(* Logix 5000 project; controller BOX_FORMING_LADDER_RS32_logixEmulate Emulate 5570 rev 32.11; software revision 32.00 *)

TASK MainTask (continuous, watchdog 500 ms) : MainProgram

MODULES
   Local : Emulate 5570 (ICP 2, rev 32.11)
      I_O : vendor 1 type 0 code 15 (ICP 3, rev 1.1, Output RPI 150 ms)
           Local:3:I   // Entradas Digitales del Controlador
           Local:3:O   // Salidas Digitales del Controlador
END_MODULES

TYPE Bloque_Instrucciones :   // Bloque de instrucciones
STRUCT
   MGSD : MOTION_INSTRUCTION;   // Arreglo donde serán almacenados los datos del bloque de función MGSD
   MGS : MOTION_INSTRUCTION;   // Arreglo donde serán almacenados los datos del bloque de función MGS
   MGSR : MOTION_INSTRUCTION;   // Arreglo donde serán almacenados los datos del bloque de función MGSR
   MAFR : MOTION_INSTRUCTION;   // Arreglo donde serán almacenados los datos del bloque de función MAFR
   MASR : MOTION_INSTRUCTION;   // Arreglo donde serán almacenados los datos del bloque de función MASR
   MSO : MOTION_INSTRUCTION;   // Arreglo donde serán almacenados los datos del bloque de función MSO
   MSF : MOTION_INSTRUCTION;   // Arreglo donde serán almacenados los datos del bloque de función MSF
   MAS : MOTION_INSTRUCTION[3];   // Arreglo donde serán almacenados los datos del bloque de función MAS
   MAH : MOTION_INSTRUCTION;   // Arreglo donde serán almacenados los datos del bloque de función MAH
   MAJ : MOTION_INSTRUCTION;   // Arreglo donde serán almacenados los datos del bloque de función MAJ
   MAG : MOTION_INSTRUCTION;   // Arreglo donde serán almacenados los datos del bloque de función MAG
   MAM : MOTION_INSTRUCTION[3];   // Arreglo donde serán almacenados los datos del bloque de función MAM
END_STRUCT
END_TYPE

VAR_GLOBAL   (* controller tags *)
   Conveyor_Belt : Bloque_Instrucciones := (MSO.FLAGS := -1577058304, MSO.EN := 1, MSO.DN := 1, MSO.STATE := 1, MSF.FLAGS := 33554432, MAS[0].FLAGS := 33554432, MAS[1].FLAGS := 33554432, MAS[2].FLAGS := 33554432, MAH.FLAGS := 33554432, MAJ.FLAGS := 570425344, MAJ.DN := 1, MAG.FLAGS := 570425344, MAG.DN := 1, MAM[0].FLAGS := 33554432, MAM[1].FLAGS := 33554432);
   Conveyor_Belt_Velocidad_Actual : REAL;   // Señal NX - Output
   DriveMSGD : MOTION_INSTRUCTION;   // Arreglo donde serán almacenados los datos del bloque de función MSGD
   Driver : Bloque_Instrucciones := (MGSD.FLAGS := 33554432, MGS.FLAGS := 33554432, MGSR.FLAGS := -1577058304, MGSR.EN := 1, MGSR.DN := 1, MAFR.FLAGS := 33554432, MASR.FLAGS := 33554432);
   DriverMAFR : MOTION_INSTRUCTION;   // Arreglo donde serán almacenados los datos del bloque de función MAFR
   DriverMASR : MOTION_INSTRUCTION;   // Arreglo donde serán almacenados los datos del bloque de función MASR
   DriverMGS : MOTION_INSTRUCTION;   // Arreglo donde serán almacenados los datos del bloque de función MGS
   DriverMGSD : MOTION_INSTRUCTION;   // Arreglo donde serán almacenados los datos del bloque de función MGSD
   DriverMGSR : MOTION_INSTRUCTION;   // Arreglo donde serán almacenados los datos del bloque de función MGSR
   DriverMSF : MOTION_INSTRUCTION;   // Arreglo donde serán almacenados los datos del bloque de función MSF
   DriverMSO : MOTION_INSTRUCTION;   // Arreglo donde serán almacenados los datos del bloque de función MSO
   Eje_X : Bloque_Instrucciones := (MSO.FLAGS := -1577058304, MSO.EN := 1, MSO.DN := 1, MSO.STATE := 1, MSF.FLAGS := 33554432, MAS[0].FLAGS := 33554432, MAS[1].FLAGS := 33554432, MAS[2].FLAGS := 33554432, MAH.FLAGS := 33554432, MAM[0].FLAGS := 33554432, MAM[1].FLAGS := 33554432, MAM[2].FLAGS := -1577058304, MAM[2].EN := 1, MAM[2].DN := 1);
   Eje_X_Posicion_Actual : REAL;   // Señal NX - Output
   Eje_Y : Bloque_Instrucciones := (MSO.FLAGS := -1577058304, MSO.EN := 1, MSO.DN := 1, MSO.STATE := 1, MSF.FLAGS := 33554432, MAS[0].FLAGS := 33554432, MAS[1].FLAGS := 33554432, MAS[2].FLAGS := 33554432, MAH.FLAGS := 33554432, MAM[0].FLAGS := 33554432, MAM[1].FLAGS := 33554432);
   Eje_Y_Posicion_Actual : REAL;   // Señal NX - Output
   Eje_Z : Bloque_Instrucciones := (MSO.FLAGS := -1577058304, MSO.EN := 1, MSO.DN := 1, MSO.STATE := 1, MSF.FLAGS := 33554432, MAS[0].FLAGS := 33554432, MAS[1].FLAGS := 33554432, MAS[2].FLAGS := 33554432, MAH.FLAGS := 33554432, MAJ.FLAGS := 637534208, MAJ.DN := 1, MAJ.IP := 1, MAG.FLAGS := 570425344, MAG.DN := 1, MAM[0].FLAGS := 33554432, MAM[1].FLAGS := 33554432);
   Eje_Z_Posicion_Actual : REAL;   // Señal NX - Output
   Fault_Reset : BOOL;
   Group_1 : MOTION_GROUP;
   Init : DINT;
   SENSOR_CAJA : BOOL;   // Señal NX - Ouput Indicator
   SPAWN_CAJA : BOOL;   // Señal NX - Output
   START_ALL : BOOL;   // BIT Destinado a la Habilitación del Sistema
   STOP_ALL : BOOL;   // BIT Destinado a la Parada del Sistema
   TESTIGO_START_ALL : ALIAS FOR Local:3:O.Data[0].0;
   TESTIGO_STOP_ALL : ALIAS FOR Local:3:O.Data[0].1;
   VIRTUAL_CONVEYOR_BELT : AXIS_VIRTUAL;   // Servomotor de la Banda Transportadora
   VIRTUAL_X_AXIS : AXIS_VIRTUAL;   // Servomotor del Eje X
   VIRTUAL_Y_AXIS : AXIS_VIRTUAL;   // Servomotor del Eje Y
   VIRTUAL_Z_AXIS : AXIS_VIRTUAL;   // Servomotor del Eje Z
END_VAR

PROGRAM MainProgram   (* main routine Main *)
VAR
   B0 : BOOL;   // Boxes Initialization Sync.
   C0 : BOOL;   // OK-INITIALIZATION
   C1 : BOOL;   // OK-CONVEYOR_BELT_IS_ON
   C2 : BOOL;   // OK-FORMADO_MOV_Y_Z
   C3 : BOOL;   // OK-FORMADO_MOV_X
   C4 : BOOL;   // OK-HOME_MOV_X_Y_Z
   C5 : BOOL;   // OK-RESET_PROCESS
   E0 : BOOL;   // INITIALIZATION
   E1 : BOOL;   // CONVEYOR_BELT_IS_ON
   E2 : BOOL;   // FORMADO_MOV_Y_Z
   E3 : BOOL;   // FORMADO_MOV_X
   E4 : BOOL;   // HOME_MOV_X_Y_Z
   E5 : BOOL;   // RESET_PROCESS
   F0 : BOOL;   // HOME_MOV_X: Transition Condition
   Fault_Reset : BOOL;   // Resetea todas las fallas/errores ocurridas en el Servo o el Driver
   H0 : BOOL;   // OK-HOME_MOV_Z: Home Flag [0]
   Servo_Off : BOOL;   // Botón físico que desabilita/desenergiza los servos
   Timer_Break_Forming : TIMER := (PRE := 400);   // Forming Break Time
   Timer_Break_Home : TIMER := (PRE := 400);   // Home Break Time
   Timer_Sensor : TIMER := (PRE := 8000);
END_VAR

ROUTINE A_Process_Setup   (* ladder *)
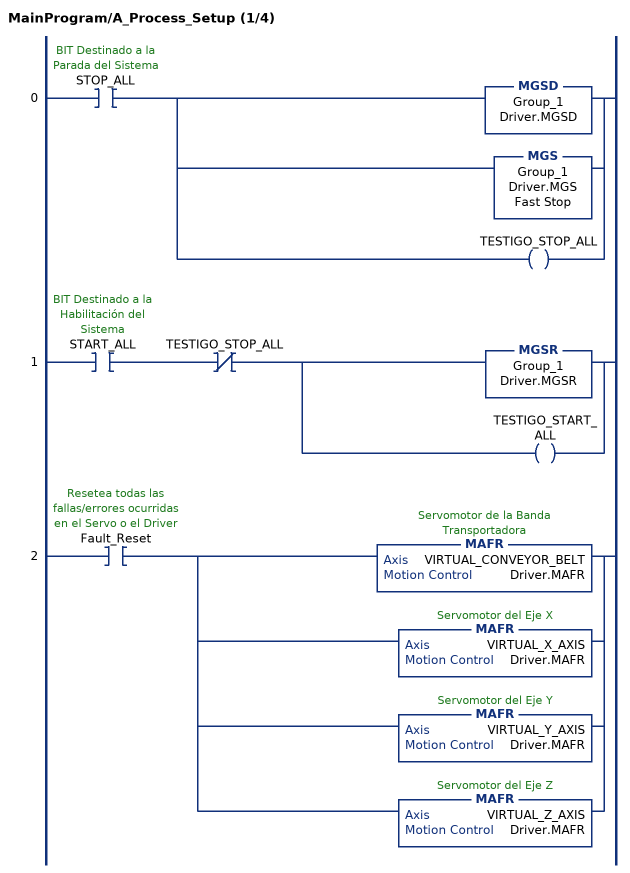
   0: XIC(STOP_ALL)[MGSD(Group_1,Driver.MGSD) ,MGS(Group_1,Driver.MGS,Fast Stop) ,OTE(TESTIGO_STOP_ALL) ];
   1: XIC(START_ALL)XIO(TESTIGO_STOP_ALL)[MGSR(Group_1,Driver.MGSR) ,OTE(TESTIGO_START_ALL) ];
   2: XIC(Fault_Reset)[MAFR(VIRTUAL_CONVEYOR_BELT,Driver.MAFR) ,MAFR(VIRTUAL_X_AXIS,Driver.MAFR) ,MAFR(VIRTUAL_Y_AXIS,Driver.MAFR) ,MAFR(VIRTUAL_Z_AXIS,Driver.MAFR) ];
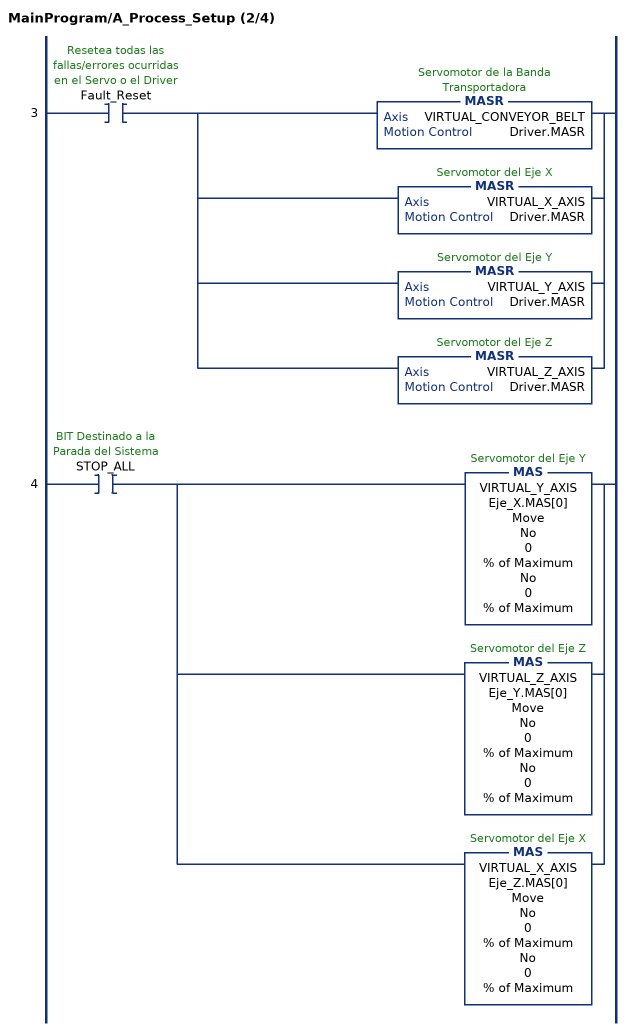
   3: XIC(Fault_Reset)[MASR(VIRTUAL_CONVEYOR_BELT,Driver.MASR) ,MASR(VIRTUAL_X_AXIS,Driver.MASR) ,MASR(VIRTUAL_Y_AXIS,Driver.MASR) ,MASR(VIRTUAL_Z_AXIS,Driver.MASR) ];
   4: XIC(STOP_ALL)[MAS(VIRTUAL_Y_AXIS,Eje_X.MAS[0],Move,No,0,% of Maximum,No,0,% of Maximum) ,MAS(VIRTUAL_Z_AXIS,Eje_Y.MAS[0],Move,No,0,% of Maximum,No,0,% of Maximum) ,MAS(VIRTUAL_X_AXIS,Eje_Z.MAS[0],Move,No,0,% of Maximum,No,0,% of Maximum) ];
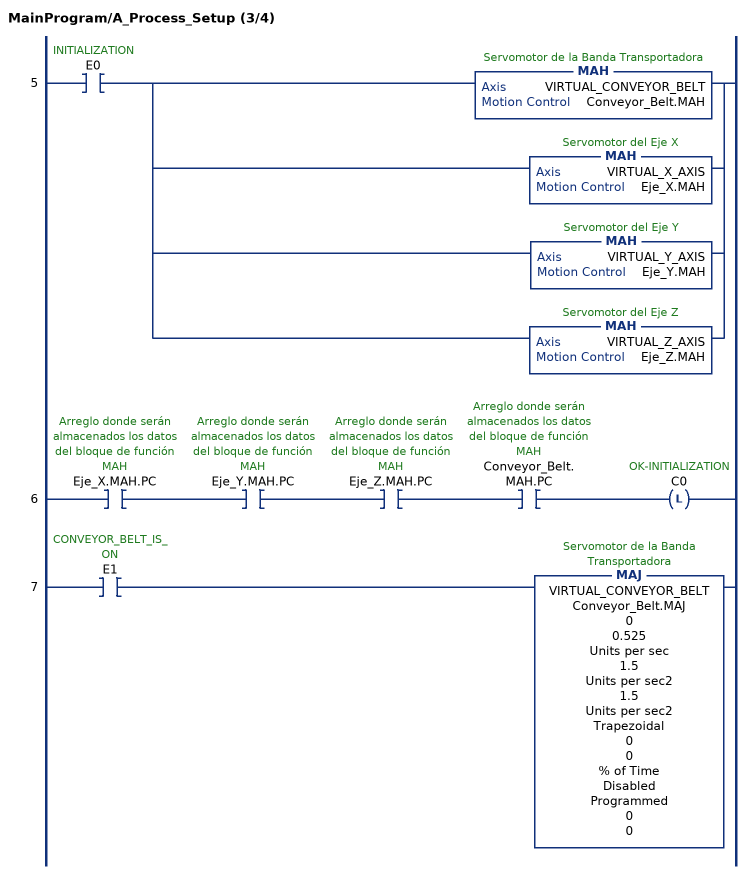
   5: XIC(E0)[MAH(VIRTUAL_CONVEYOR_BELT,Conveyor_Belt.MAH) ,MAH(VIRTUAL_X_AXIS,Eje_X.MAH) ,MAH(VIRTUAL_Y_AXIS,Eje_Y.MAH) ,MAH(VIRTUAL_Z_AXIS,Eje_Z.MAH) ];
   6: XIC(Eje_X.MAH.PC)XIC(Eje_Y.MAH.PC)XIC(Eje_Z.MAH.PC)XIC(Conveyor_Belt.MAH.PC)OTL(C0);
   7: XIC(E1)MAJ(VIRTUAL_CONVEYOR_BELT,Conveyor_Belt.MAJ,0,0.525,Units per sec,1.5,Units per sec2,1.5,Units per sec2,Trapezoidal,0,0,% of Time,Disabled,Programmed,0,0);
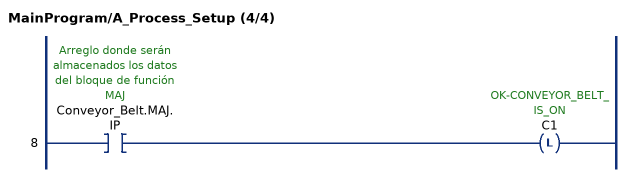
   8: XIC(Conveyor_Belt.MAJ.IP)OTL(C1);
END_ROUTINE

ROUTINE B_Process_Formado   (* ladder *)
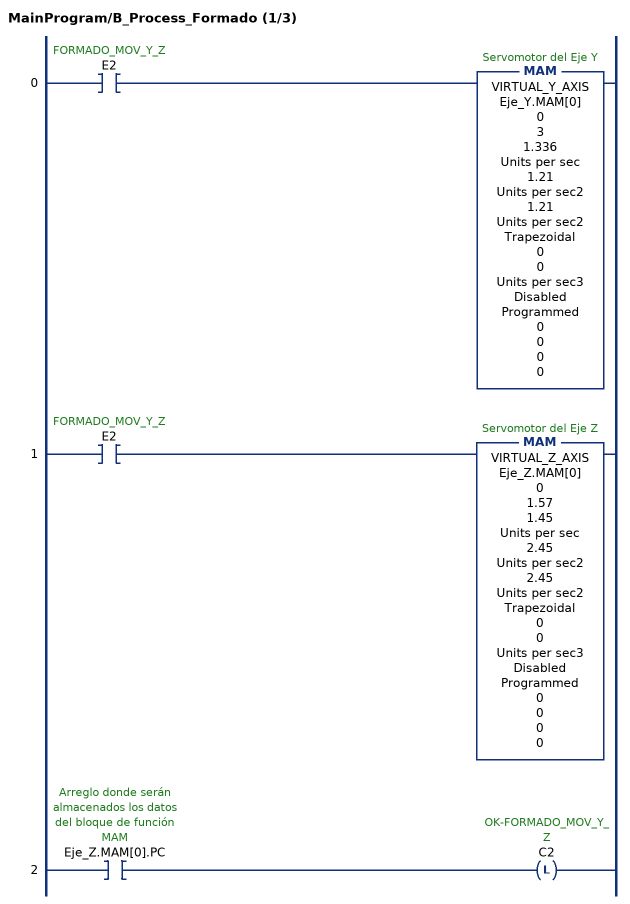
   0: XIC(E2)MAM(VIRTUAL_Y_AXIS,Eje_Y.MAM[0],0,3,1.336,Units per sec,1.21,Units per sec2,1.21,Units per sec2,Trapezoidal,0,0,Units per sec3,Disabled,Programmed,0,0,0,0);
   1: XIC(E2)MAM(VIRTUAL_Z_AXIS,Eje_Z.MAM[0],0,1.57,1.45,Units per sec,2.45,Units per sec2,2.45,Units per sec2,Trapezoidal,0,0,Units per sec3,Disabled,Programmed,0,0,0,0);
   2: XIC(Eje_Z.MAM[0].PC)OTL(C2);
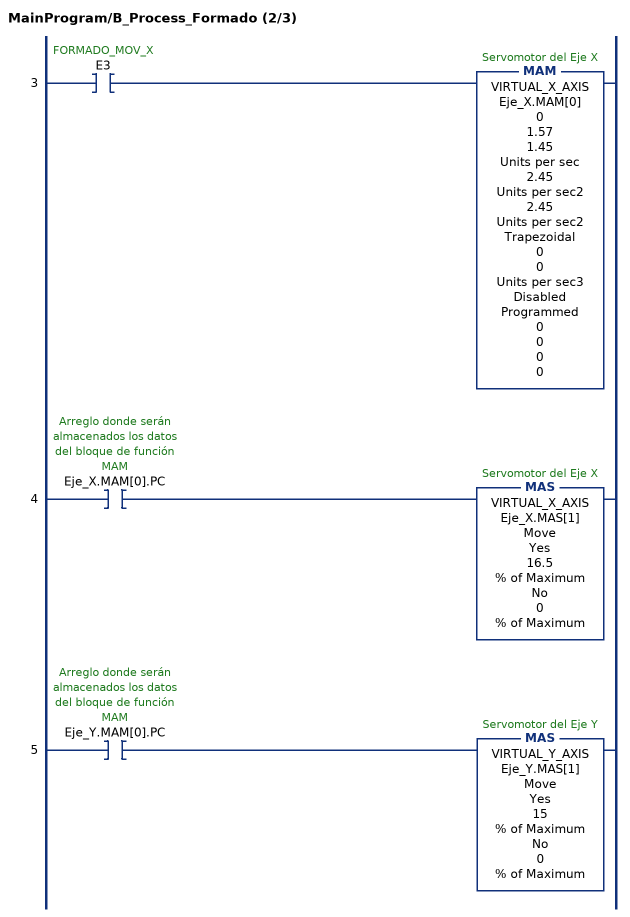
   3: XIC(E3)MAM(VIRTUAL_X_AXIS,Eje_X.MAM[0],0,1.57,1.45,Units per sec,2.45,Units per sec2,2.45,Units per sec2,Trapezoidal,0,0,Units per sec3,Disabled,Programmed,0,0,0,0);
   4: XIC(Eje_X.MAM[0].PC)MAS(VIRTUAL_X_AXIS,Eje_X.MAS[1],Move,Yes,16.5,% of Maximum,No,0,% of Maximum);
   5: XIC(Eje_Y.MAM[0].PC)MAS(VIRTUAL_Y_AXIS,Eje_Y.MAS[1],Move,Yes,15,% of Maximum,No,0,% of Maximum);
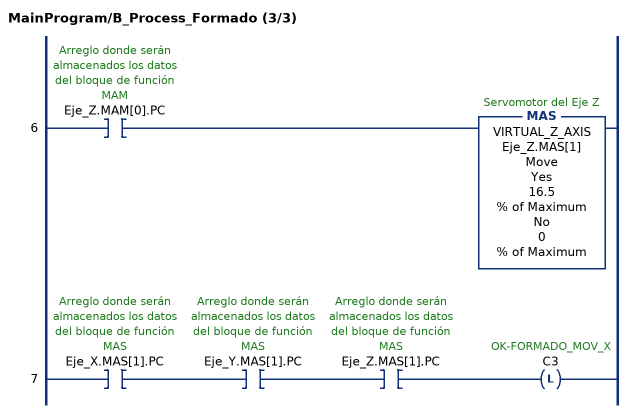
   6: XIC(Eje_Z.MAM[0].PC)MAS(VIRTUAL_Z_AXIS,Eje_Z.MAS[1],Move,Yes,16.5,% of Maximum,No,0,% of Maximum);
   7: XIC(Eje_X.MAS[1].PC)XIC(Eje_Y.MAS[1].PC)XIC(Eje_Z.MAS[1].PC)OTL(C3);
END_ROUTINE

ROUTINE C_Process_Home   (* ladder *)
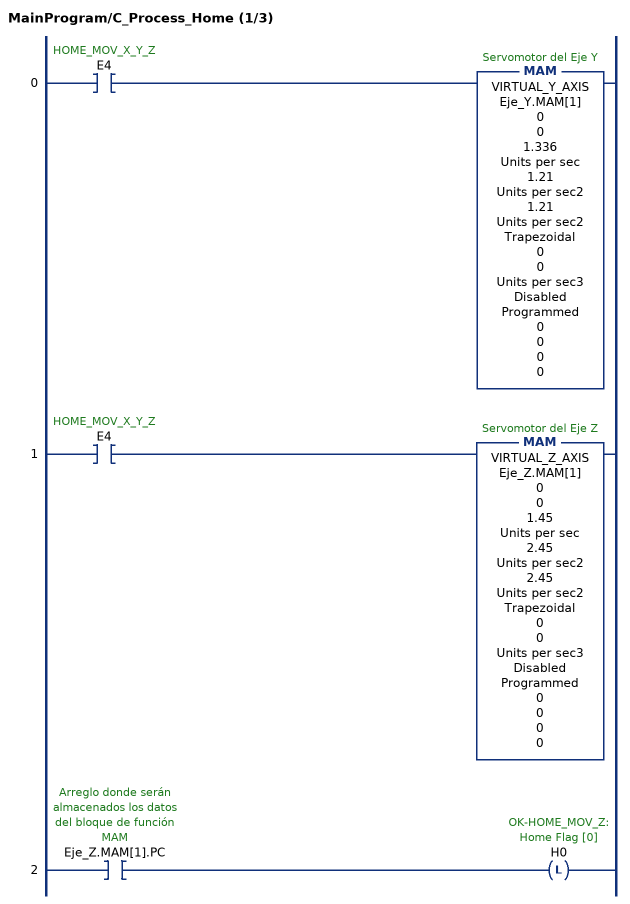
   0: XIC(E4)MAM(VIRTUAL_Y_AXIS,Eje_Y.MAM[1],0,0,1.336,Units per sec,1.21,Units per sec2,1.21,Units per sec2,Trapezoidal,0,0,Units per sec3,Disabled,Programmed,0,0,0,0);
   1: XIC(E4)MAM(VIRTUAL_Z_AXIS,Eje_Z.MAM[1],0,0,1.45,Units per sec,2.45,Units per sec2,2.45,Units per sec2,Trapezoidal,0,0,Units per sec3,Disabled,Programmed,0,0,0,0);
   2: XIC(Eje_Z.MAM[1].PC)OTL(H0);
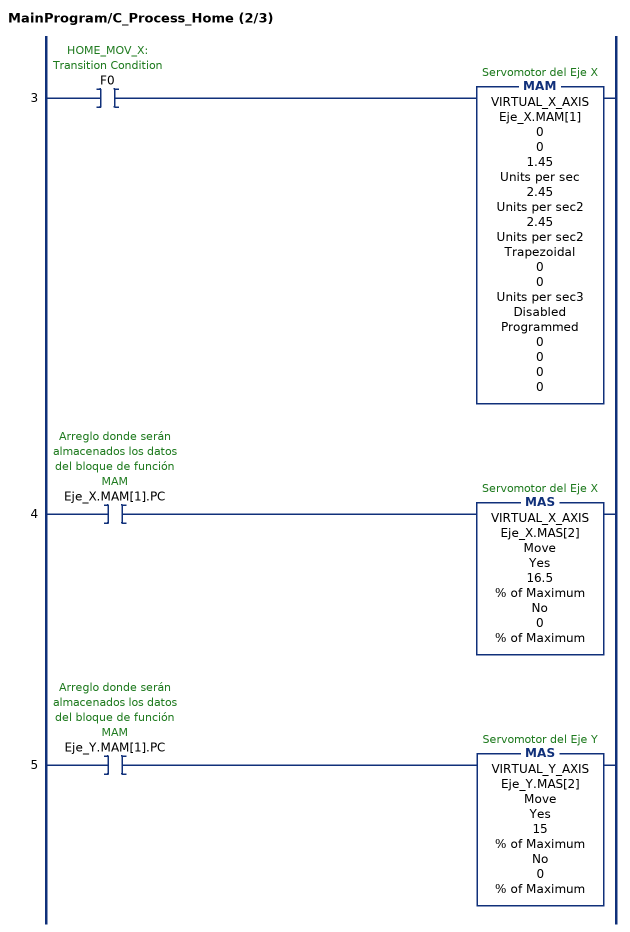
   3: XIC(F0)MAM(VIRTUAL_X_AXIS,Eje_X.MAM[1],0,0,1.45,Units per sec,2.45,Units per sec2,2.45,Units per sec2,Trapezoidal,0,0,Units per sec3,Disabled,Programmed,0,0,0,0);
   4: XIC(Eje_X.MAM[1].PC)MAS(VIRTUAL_X_AXIS,Eje_X.MAS[2],Move,Yes,16.5,% of Maximum,No,0,% of Maximum);
   5: XIC(Eje_Y.MAM[1].PC)MAS(VIRTUAL_Y_AXIS,Eje_Y.MAS[2],Move,Yes,15,% of Maximum,No,0,% of Maximum);
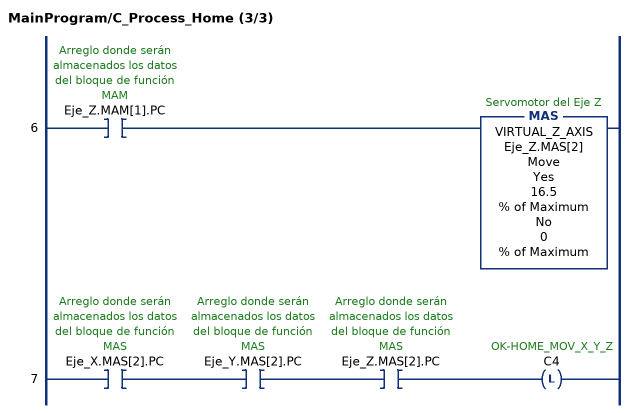
   6: XIC(Eje_Z.MAM[1].PC)MAS(VIRTUAL_Z_AXIS,Eje_Z.MAS[2],Move,Yes,16.5,% of Maximum,No,0,% of Maximum);
   7: XIC(Eje_X.MAS[2].PC)XIC(Eje_Y.MAS[2].PC)XIC(Eje_Z.MAS[2].PC)OTL(C4);
END_ROUTINE

ROUTINE D_Process_Reset   (* ladder *)
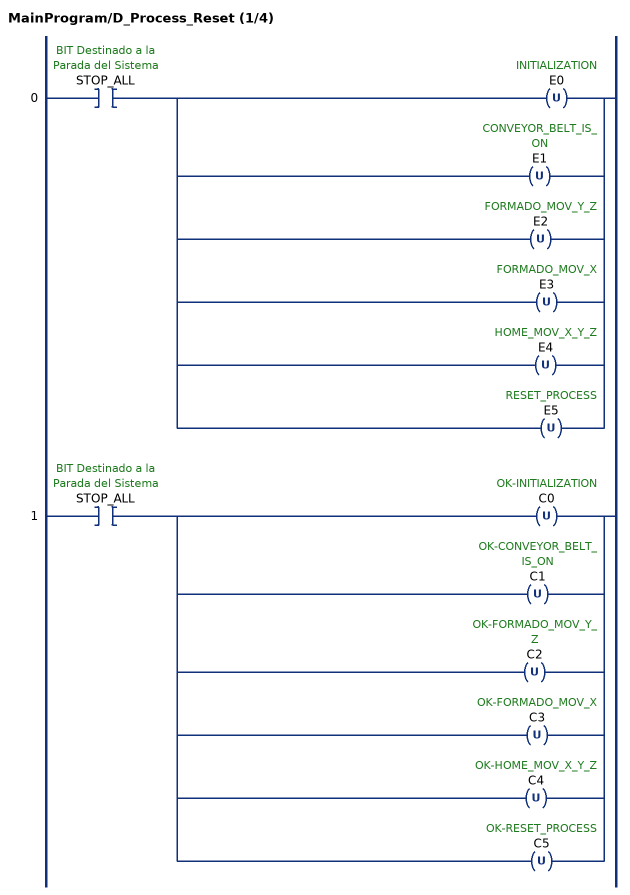
   0: XIC(STOP_ALL)[OTU(E0) ,OTU(E1) ,OTU(E2) ,OTU(E3) ,OTU(E4) ,OTU(E5) ];
   1: XIC(STOP_ALL)[OTU(C0) ,OTU(C1) ,OTU(C2) ,OTU(C3) ,OTU(C4) ,OTU(C5) ];
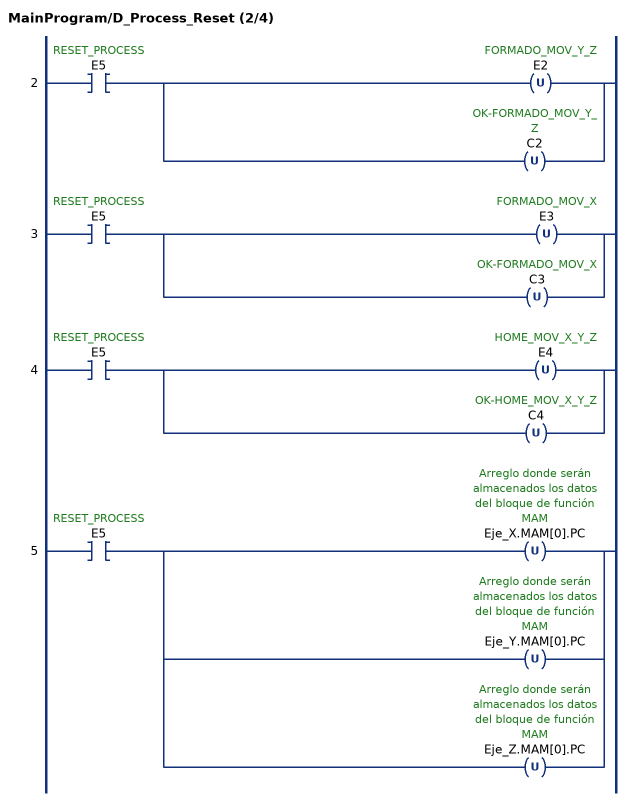
   2: XIC(E5)[OTU(E2) ,OTU(C2) ];
   3: XIC(E5)[OTU(E3) ,OTU(C3) ];
   4: XIC(E5)[OTU(E4) ,OTU(C4) ];
   5: XIC(E5)[OTU(Eje_X.MAM[0].PC) ,OTU(Eje_Y.MAM[0].PC) ,OTU(Eje_Z.MAM[0].PC) ];
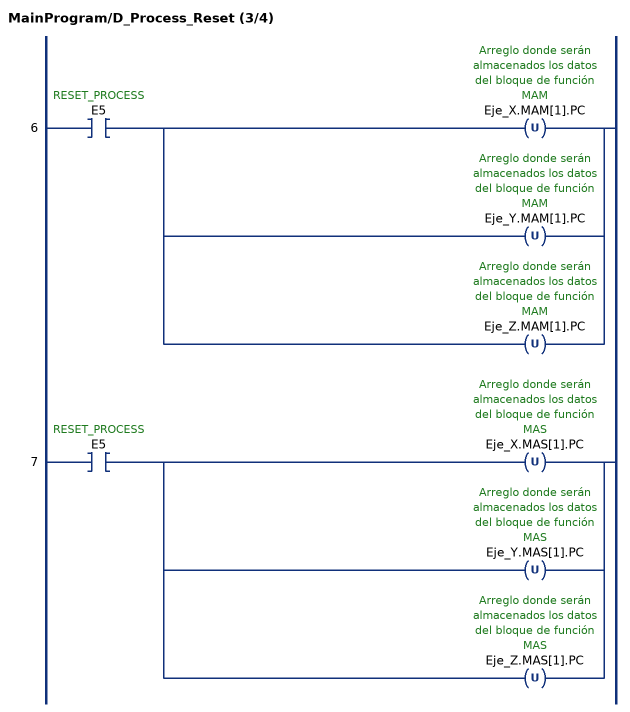
   6: XIC(E5)[OTU(Eje_X.MAM[1].PC) ,OTU(Eje_Y.MAM[1].PC) ,OTU(Eje_Z.MAM[1].PC) ];
   7: XIC(E5)[OTU(Eje_X.MAS[1].PC) ,OTU(Eje_Y.MAS[1].PC) ,OTU(Eje_Z.MAS[1].PC) ];
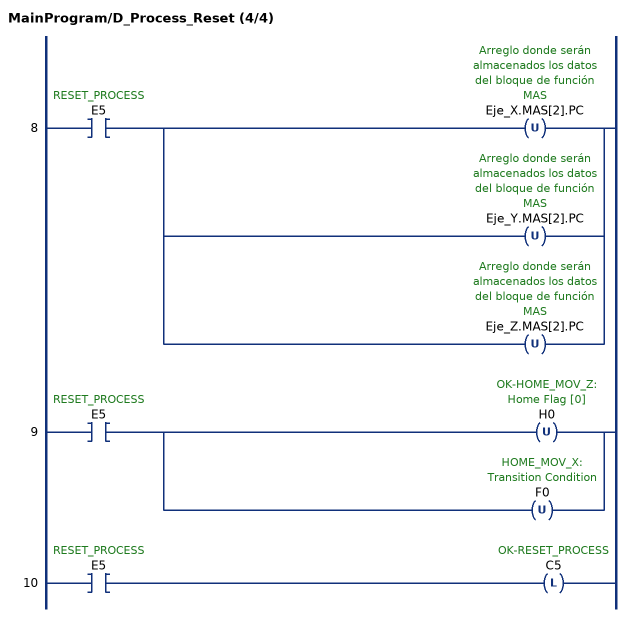
   8: XIC(E5)[OTU(Eje_X.MAS[2].PC) ,OTU(Eje_Y.MAS[2].PC) ,OTU(Eje_Z.MAS[2].PC) ];
   9: XIC(E5)[OTU(H0) ,OTU(F0) ];
   10: XIC(E5)OTL(C5);
END_ROUTINE

ROUTINE Main   (* ladder *)
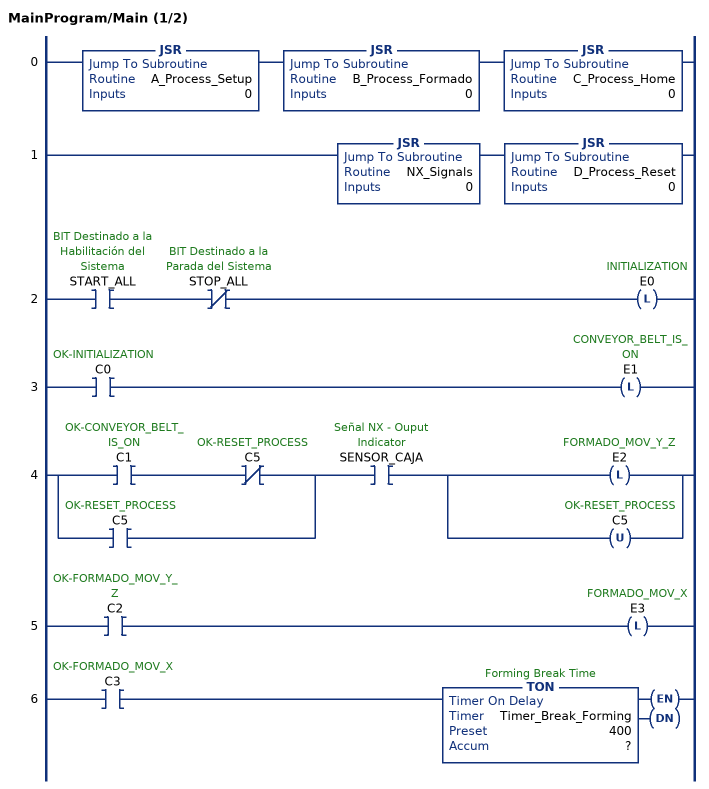
   0: JSR(A_Process_Setup,0)JSR(B_Process_Formado,0)JSR(C_Process_Home,0);
   1: JSR(NX_Signals,0)JSR(D_Process_Reset,0);
   2: XIC(START_ALL)XIO(STOP_ALL)OTL(E0);
   3: XIC(C0)OTL(E1);
   4: [XIC(C1) XIO(C5) ,XIC(C5) ]XIC(SENSOR_CAJA)[OTL(E2) ,OTU(C5) ];
   5: XIC(C2)OTL(E3);
   6: XIC(C3)TON(Timer_Break_Forming,?,?);
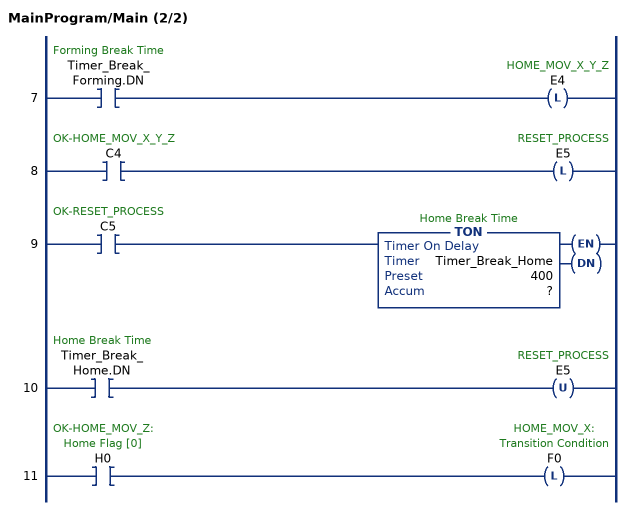
   7: XIC(Timer_Break_Forming.DN)OTL(E4);
   8: XIC(C4)OTL(E5);
   9: XIC(C5)TON(Timer_Break_Home,?,?);
   10: XIC(Timer_Break_Home.DN)OTU(E5);
   11: XIC(H0)OTL(F0);
END_ROUTINE

ROUTINE NX_Signals   (* ladder *)
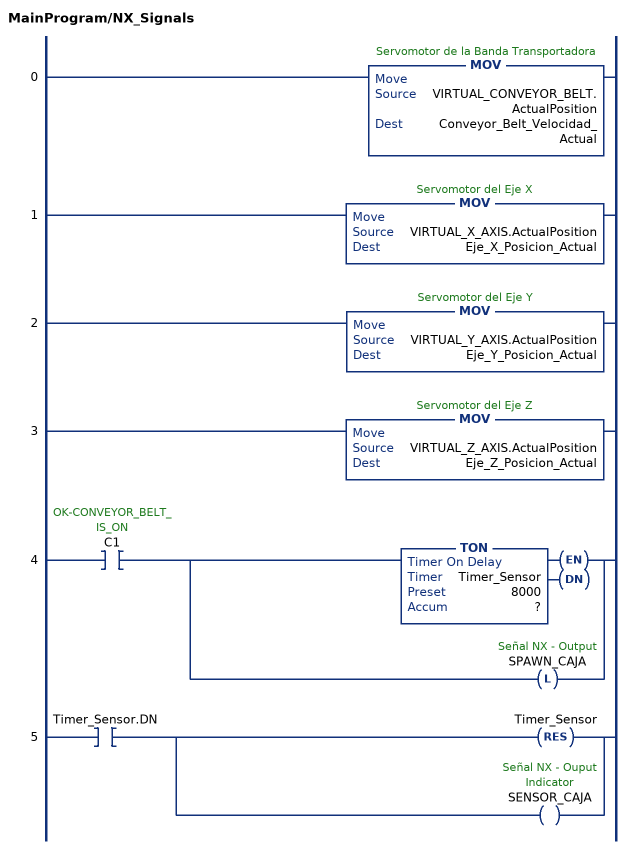
   0: MOV(VIRTUAL_CONVEYOR_BELT.ActualPosition,Conveyor_Belt_Velocidad_Actual);
   1: MOV(VIRTUAL_X_AXIS.ActualPosition,Eje_X_Posicion_Actual);
   2: MOV(VIRTUAL_Y_AXIS.ActualPosition,Eje_Y_Posicion_Actual);
   3: MOV(VIRTUAL_Z_AXIS.ActualPosition,Eje_Z_Posicion_Actual);
   4: XIC(C1)[TON(Timer_Sensor,?,?) ,OTL(SPAWN_CAJA) ];
   5: XIC(Timer_Sensor.DN)[RES(Timer_Sensor) ,OTE(SENSOR_CAJA) ];
END_ROUTINE
END_PROGRAM
